FUNCTION_BLOCK FB_HomeGantry
VAR_INPUT
	Enable : BOOL;
	KidID : INT;
	HomeStart : BOOL;
	OffHome : BOOL;
	KidStart : DINT;
	CaseNum : DINT;
	PrevVel : DINT; 
END_VAR
VAR_OUTPUT
END_VAR
VAR

END_VAR

IF  KidID = 0 THEN RETURN; END_IF

IF NOT enable OR MAIN.GlobalEstopActive THEN
	main.Kid[kidid].TargetPos := main.Kid[kidID].currentPosition;
END_IF

IF HomeStart THEN
	PrevVel := MAIN.Kid[KidID].modeVel;
	KidStart := MAIN.Kid[KidID].currentPosition;
	MAIN.Kid[KidID].CheckIn.HomeOperation_Active := TRUE;
	HomeStart := FALSE;
	OffHome := FALSE;
	CaseNum := 0;
END_IF


CASE CaseNum OF
	0:
		IF KidID = 1 THEN MAIN.Kid[KidID].TargetPos := KidStart + 100; END_IF
		IF KidID = 3 THEN MAIN.Kid[KidID].TargetPos := KidStart - 100; END_IF
		IF KidID = 2 THEN MAIN.Kid[KidID].TargetPos := KidStart + 100; END_IF
		IF KidID = 4 THEN MAIN.Kid[KidID].TargetPos := KidStart + 100; END_IF
		
		MAIN.Kid[KidID].modeVel := MAIN.Kid[KidID].HomeSpeed;
		IF MAIN.Kid[KidID].CheckIn.HomeActivated  THEN 
			CaseNum := CaseNum + 1; 
		ELSIF ABS(MAIN.Kid[KidID].currentPosition - MAIN.Kid[KidID].TargetPos) < 10 THEN 
			CaseNum := CaseNum + 2; 
		END_IF
	1: 
		IF KidID = 1 THEN MAIN.Kid[KidID].TargetPos := MAIN.Kid[KidID].currentPosition + 100; END_IF
		IF KidID = 3 THEN MAIN.Kid[KidID].TargetPos := MAIN.Kid[KidID].currentPosition - 100; END_IF
		IF KidID = 2 THEN MAIN.Kid[KidID].TargetPos := KidStart + 1000; END_IF
		IF KidID = 4 THEN MAIN.Kid[KidID].TargetPos := KidStart + 1000; END_IF
		
		IF (KidID = 1 OR KidId = 3) AND NOT MAIN.Kid[KidID].CheckIn.HomeActivated OR MAIN.GantryCollision  THEN CaseNum := CaseNum + 1; END_IF
		IF (KidID = 2 OR KidId = 4) AND MAIN.Kid[KidID].CheckIn.Hard_Limit_Tripped  THEN  CaseNum := CaseNum + 1; END_IF
	2: 
		IF KidID = 3 THEN MAIN.Kid[KidID].TargetPos := MAIN.Kid[KidID].currentPosition + 100; END_IF
		IF KidID = 1 THEN MAIN.Kid[KidID].TargetPos := MAIN.Kid[KidID].currentPosition - 100; END_IF
		
		IF (KidID = 1 OR KidID = 3) AND MAIN.Kid[KidID].CheckIn.HomeActivated  THEN 
			MAIN.Kid[KidID].modeVel := MAIN.Kid[KidID].HomeSpeed/3;
			CaseNum := CaseNum + 1;
		ELSIF (KidID = 2 OR KidID = 4) AND MAIN.Kid[KidID].CheckIn.Hard_Limit_Tripped THEN
			MAIN.Kid[KidID].CheckIn.HomeOperation_Active := FALSE;
			CaseNum := CaseNum + 2;
		END_IF
			
	3: 
		IF KidID = 3 THEN MAIN.Kid[KidID].TargetPos := MAIN.Kid[KidID].currentPosition + 100; END_IF
		IF KidID = 1 THEN MAIN.Kid[KidID].TargetPos := MAIN.Kid[KidID].currentPosition - 100; END_IF
		IF NOT MAIN.Kid[KidID].CheckIn.HomeActivated  THEN 
			MAIN.Kid[KidID].CheckIn.HomeOperation_Active := FALSE;
			CaseNum := CaseNum + 1;
		END_IF
	4: 	
		//IF KidID = 1 THEN MAIN.Kid[KidID].TargetPos := 0; END_IF;
	   //	IF KidID = 3 THEN MAIN.Kid[KidID].TargetPos := 3295; END_IF;
		//IF  ABS(MAIN.Kid[KidID].currentPosition - MAIN.Kid[KidID].TargetPos) < 10 THEN
			MAIN.Kid[KidID].TargetPos := MAIN.Kid[KidID].currentPosition;
			Enable := FALSE;
				Main.Kid[kidid].modeVel := DINT_TO_UINT(prevVel);
			KidID := 0;
			
		
		//	MAIN.Kid[KidID].RMT_DeadManPressed := FALSE;
		//	CaseNum := CaseNum + 1;
		//END_IF
	5: 
	
END_CASE

END_FUNCTION_BLOCK

(* stored: Version 1.1.0.1, ProductVersion 3.1.4022.3
   POU FB_HomeGantry: Id {967aac62-0684-45fa-82b7-1e8dbf7ade35}, SpecialFunc None *)
